# EPICS StreamDevice protocol: TC110.proto
Terminator = CR;

#001 Heating
readHeating {out "1230000102=?%+<sum8>";in "1231000106%{000000|111111}%+<sum8>";}
setHeating {out "1231000106%{000000|111111}%+<sum8>";in "1231000106%{000000|111111}%+<sum8>";}

#002 Standby
readStandby {out "1230000202=?%+<sum8>";in "1231000206%{000000|111111}%+<sum8>";}
setStandby {out "1231000206%{000000|111111}%+<sum8>";in "1231000206%{000000|111111}%+<sum8>";}

#012 Enable venting
readenablevent {out "1230001202=?%+<sum8>";in "1231001206%{000000|111111}%+<sum8>";}
setenablevent {out "1231001206%{000000|111111}%+<sum8>";in "1231001206%{000000|111111}%+<sum8>";}

#023 Motor Pump
readmotorpump {out "1230002302=?%+<sum8>";in "1231002306%{000000|111111}%+<sum8>";}
setmotorpump {out "1231002306%{000000|111111}%+<sum8>";in "1231002306%{000000|111111}%+<sum8>";}

#025 Operation mode backing pump
readOpModeBKP {out "1230002502=?%+<sum8>";in "1231002503%3.3d%+<sum8>";}
setmotorpump {out "1231002503%3.3d%+<sum8>";in "1231002503%3.3d%+<sum8>";}

#026 Rotation speed setting mode
readSpdSetMode {out "1230002602=?%+<sum8>";in "1231002603%3.3d%+<sum8>";}
setSpdSetMode {out "1231002603%3.3d%+<sum8>";in "1231002603%3.3d%+<sum8>";}

#027 gas mode
readgasmode {out "1230002702=?%+<sum8>";in "1231002703%3.3d%+<sum8>";}
setgasmode {out "1231002703%3.3d%+<sum8>";in "1231002703%3.3d%+<sum8>";}

#030 Venting mode
readventingmode {out "1230003002=?%+<sum8>";in "1231003003%3.3d%+<sum8>";}
setventingmode {out "1231003003%3.3d%+<sum8>";in "1231003003%3.3d%+<sum8>";}

#050 Sealing gas
readsealinggas {out "1230005002=?%+<sum8>"; in "1231005006%{000000|111111}%+<sum8>";}
setsealinggas {out "1231005006%{000000|111111}%+<sum8>"; in "1231005006%{000000|111111}%+<sum8>";}

#060 Control via interface
readCtrlVialnt {out "1230006002=?%+<sum8>";in "1231006003%3.3d%+<sum8>";}
setCtrlVialnt {out "1231006003%3.3d%+<sum8>";in "1231006003%3.3d%+<sum8>";}

#061 Interface selection locked
readIntSelLckd {out "1230006102=?%+<sum8>";in "1231006106%{000000|111111}%+<sum8>";}
setIntSelLckd {out "1231006106%{000000|111111}%+<sum8>";in "1231006106%{000000|111111}%+<sum8>";}

#300 Remote priority
readRemotePrio {out "1230030002=?%+<sum8>";in "1231030006%{000000|111111}%+<sum8>";}
setRemotePrio {out "1231030006%{000000|111111}%+<sum8>";in "1231030006%{000000|111111}%+<sum8>";}

#304 Overtemperature electronic drive unit
readOvTempElec {out "1230030402=?%+<sum8>"; in "1231030406%{000000|111111}%+<sum8>";}

#305 Overtemperature pump
readOvTempPump {out "1230030502=?%+<sum8>"; in "1231030506%{000000|111111}%+<sum8>";}

#306 Target speed reached
readsetSpdAtt {out "1230030602=?%+<sum8>"; in "1231030606%{000000|111111}%+<sum8>";}

#307 Pump accelerating
readPumpAccel {out "1230030702=?%+<sum8>"; in "1231030706%{000000|111111}%+<sum8>";}

#308 Actual rotation speed
readsetRotSpdHz {out "1230030802=?%+<sum8>"; in "1231030806%6.6d%+<sum8>";}

#309 Actual rotation speed
readActualSpdHz {out "1230030902=?%+<sum8>"; in "1231030906%6.6d%+<sum8>";}

#310 Drive current
readDrvCurrent {out "1230031002=?%+<sum8>"; in "1231031006%6.6d%+<sum8>";}

#313 Drive voltage
readDrvVoltage {out "1230031302=?%+<sum8>"; in "1231031306%6.6d%+<sum8>";}

#315 Nominal Spd
readNominalSpd {out "1230031502=?%+<sum8>"; in "1231031506%6.6d%+<sum8>";}

#316 Drive power
readDrvPower {out "1230031602=?%+<sum8>"; in "1231031606%6.6d%+<sum8>";}

#326 Temperature electronics
readTempElec {out "1230032602=?%+<sum8>"; in "1231032606%6.6d%+<sum8>";}

#330 Temperature Pump bottom part
readTempPumpBot {out "1230033002=?%+<sum8>"; in "1231033006%6.6d%+<sum8>";}

#397 Actual rotation speed
readsetRotSpdrpm {out "1231039702=?%+<sum8>"; in "1231039706%6.6d%+<sum8>";}

#398 Actual rotation speed
readActualSpdrpm {out "1230039802=?%+<sum8>"; in "1231039806%6.6d%+<sum8>";}

#399 Nominal Speed
readNominalSpd {out "1230039902=?%+<sum8>"; in "1231039906%6.6d%+<sum8>";}
